// TIA Portal V20 export
DATA_BLOCK "Config"   // DB180
// stored: Access Published, MemoryReserve 100, Namespace Unit1.Em4
   VAR
      em : "LAF_typeEmConfiguration";   // Configuration of EM Parameters
      axis : Array[0.._.U1EM4_NO_OF_AXES] of DB_ANY;
      cmSideTapeSafetyPin : "LBC_typeDigitalSignalConfiguration";
      cmSideTapeJRDetect : "LBC_typeDigitalSignalConfiguration";
      cmSideTapeDiameter : "LBC_typeDigitalSignalConfiguration";
   END_VAR
   VAR RETAIN
      cmSideTapeFixStageAxisX : "LBC_typeAxis64PosConfiguration";
      cmSideTapeFixStageAxisC : "LBC_typeAxis64PosConfiguration";
      cmSideTapeAttachmentAxisX : "LBC_typeAxis64PosConfiguration";
      cmSideTapeAttachmentAxisY : "LBC_typeAxis64PosConfiguration";
   END_VAR
   VAR
      cmSideTapeLoadingDownUp : "LBC_typeTwoWayActuatorConfiguration";
      cmSideTapeLoadingClampOpenClose : "LBC_typeTwoWayActuatorConfiguration";
      cmSideTapeCutterBwdFwd : "LBC_typeTwoWayActuatorConfiguration";
      cmSideTapeCutterClampBwdFwd : "LBC_typeTwoWayActuatorConfiguration";
      cmSideTapeTensionBwdFwd : "LBC_typeTwoWayActuatorConfiguration";
      cmSideTapeAttachmentLeftBwdFwd : "LBC_typeTwoWayActuatorConfiguration";
      cmSideTapeAttachmentRightBwdFwd : "LBC_typeTwoWayActuatorConfiguration";
      cmSideTapeAttachmentBtmBwdFwd : "LBC_typeTwoWayActuatorConfiguration";
      cmSideTapeFixStageClampOpenClose : "LBC_typeTwoWayActuatorConfiguration";
      cmSideTapeAttachment1TopVaccumOffOn : "LBC_typeTwoWayActuatorConfiguration";
      cmSideTapeAttachment1BtmVaccumOffOn : "LBC_typeTwoWayActuatorConfiguration";
      cmSideTapeAttachment2TopVaccumOffOn : "LBC_typeTwoWayActuatorConfiguration";
      cmSideTapeAttachment2BtmVaccumOffOn : "LBC_typeTwoWayActuatorConfiguration";
      cmQrHandyReader : "LER_typeDM8700Configuration";
      softcam : Struct
         SideTapeFixStageAxisX : "LER_typeSoftCamInterface";
         SideTapeFixStageAxisC : "LER_typeSoftCamInterface";
         SideTapeAttachmentAxisX : "LER_typeSoftCamInterface";
         SideTapeAttachmentAxisY { S7_SetPoint := 'True'} : "LER_typeSoftCamInterface";
      END_STRUCT;
   END_VAR
BEGIN
   em.referenceDesignator.parent := WSTRING#'U1';
   em.referenceDesignator.relative := WSTRING#'EM2';
   cmSideTapeFixStageAxisX.referenceDesignator := WSTRING#'Fix Stage X-Axis';
   cmSideTapeFixStageAxisC.referenceDesignator := WSTRING#'Fix Stage C-Axis';
   cmSideTapeAttachmentAxisX.referenceDesignator := WSTRING#'Attachment X-Axis';
   cmSideTapeAttachmentAxisY.referenceDesignator := WSTRING#'Attachment Y-Axis';
   cmSideTapeLoadingDownUp.referenceDesignator := WSTRING#'S.TAPE LOADING';
   cmSideTapeLoadingDownUp.monitoringDiscrepancy := T#5s;
   cmSideTapeLoadingClampOpenClose.referenceDesignator := WSTRING#'S.TAPE LOADING CLAMP';
   cmSideTapeLoadingClampOpenClose.monitoringDiscrepancy := T#5s;
   cmSideTapeCutterBwdFwd.referenceDesignator := WSTRING#'S.TAPE CUTTER';
   cmSideTapeCutterBwdFwd.monitoringDiscrepancy := T#5s;
   cmSideTapeCutterClampBwdFwd.referenceDesignator := WSTRING#'S.TAPE CUTTER CLAMP';
   cmSideTapeCutterClampBwdFwd.monitoringDiscrepancy := T#5s;
   cmSideTapeTensionBwdFwd.referenceDesignator := WSTRING#'S.TAPE TENSION';
   cmSideTapeTensionBwdFwd.monitoringDiscrepancy := T#5s;
   cmSideTapeAttachmentLeftBwdFwd.referenceDesignator := WSTRING#'S.TAPE ATTACH LEFT';
   cmSideTapeAttachmentLeftBwdFwd.monitoringDiscrepancy := T#5s;
   cmSideTapeAttachmentRightBwdFwd.referenceDesignator := WSTRING#'S.TAPE ATTACH RIGHT';
   cmSideTapeAttachmentRightBwdFwd.monitoringDiscrepancy := T#5s;
   cmSideTapeAttachmentBtmBwdFwd.referenceDesignator := WSTRING#'S.TAPE ATTACH BTM';
   cmSideTapeAttachmentBtmBwdFwd.monitoringDiscrepancy := T#5s;
   cmSideTapeFixStageClampOpenClose.referenceDesignator := WSTRING#'JR FIX STAGE CLAMP';
   cmSideTapeFixStageClampOpenClose.monitoringDiscrepancy := T#5s;
   cmSideTapeAttachment1TopVaccumOffOn.referenceDesignator := WSTRING#'ATTACH LEFT TOP VACUUM';
   cmSideTapeAttachment1TopVaccumOffOn.monitoringDiscrepancy := T#5s;
   cmSideTapeAttachment1BtmVaccumOffOn.referenceDesignator := WSTRING#'ATTACH LEFT BTM VACUUM';
   cmSideTapeAttachment1BtmVaccumOffOn.monitoringDiscrepancy := T#5s;
   cmSideTapeAttachment2TopVaccumOffOn.referenceDesignator := WSTRING#'ATTACH RIGHT TOP VACUUM';
   cmSideTapeAttachment2TopVaccumOffOn.monitoringDiscrepancy := T#5s;
   cmSideTapeAttachment2BtmVaccumOffOn.referenceDesignator := WSTRING#'ATTACH RIGHT BTM VACUUM';
   cmSideTapeAttachment2BtmVaccumOffOn.monitoringDiscrepancy := T#5s;
END_DATA_BLOCK
